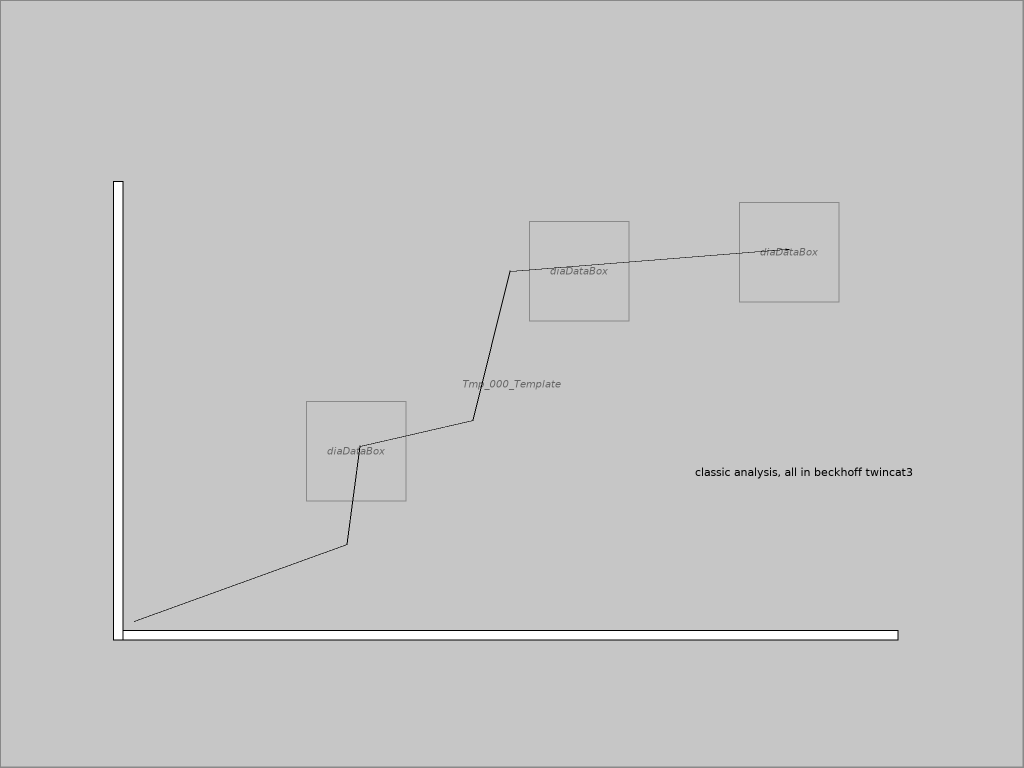
VISUALIZATION Dat_550_DataAxis  // 1024x768
    Frame (0,0 1024x768)
        shows Tmp_000_Template(header := gHMIData.hmiHeader)
    Frame (306,401 100x100)
        shows diaDataBox()
    Frame (529,221 100x100)
        shows diaDataBox()
    Frame (739,202 100x100)
        shows diaDataBox()
    Rectangle (113,630 785x10)
    Rectangle (113,181 10x459)
    Polyline (134,621) (347,544) (360,446) (473,420) (510,271) (786,249) (789,249)
    Label (667,461 274x23), "classic analysis, all in beckhoff twincat3"
END_VISUALIZATION

(* stored: Version 1.1.0.1, ProductVersion 3.1.4024.11
   Visu Dat_550_DataAxis: Id {bdd6f013-ccbd-0e76-355e-144e569364ab} *)
